(* Logix 5000 project; controller Pensador vendor 1 type 14 code 15 rev 20.11; software revision 20.04 *)

TASK MainTask (continuous, watchdog 500 ms) : MainProgram

MODULES
   Local : vendor 1 type 14 code 15 (SoftLogixController 2, rev 20.11)
      Ethernet : vendor 1 type 12 code 135 (SoftLogixVB 3, Ethernet 192.168.0.160, rev 20.1)
END_MODULES

VAR_GLOBAL   (* controller tags *)
   Acender_Led_Amarelo : BOOL := 1;
   Acender_Led_Azul : BOOL := 1;
   Acender_Led_Branco : BOOL := 1;
   Acender_Led_Transparente : BOOL;
   Acender_Led_Verde : BOOL := 1;
   Acender_Led_Vermelho : BOOL := 1;
   Acionamentos : DINT := 52;
   aguarde : BOOL;
   Alarme : DINT;
   Alinhador : STRING[20] := ([0] := 'Azul', [1] := 'Desliga_Azul', [2] := 'Vermelho', [3] := 'Desliga_Vermelho', [4] := 'Transparente', [5] := 'Desliga_Transparente', [6] := 'Amarelo', [7] := 'Desliga_Amarelo', [8] := 'Verde', [9] := 'Desliga_Verde');
   Botao_B01 : BOOL;
   Botao_B02 : BOOL := 1;
   Botao_B03 : BOOL;
   Botao_Pressionado : BOOL;
   Camera : STRING;
   CameraInt : DINT;
   Chamada_de_Voz : BOOL;
   Chave : SINT;
   Comparador : STRING := 'Ligar LED azul';
   Comparador2 : STRING := 'desligar led azul';
   Comparador3 : STRING := 'Ligar LED verde';
   Comparador4 : STRING := 'desligar led Verde';
   Comparador5 : STRING := 'Ligar LED branco';
   Comparador6 : STRING := 'desligar LED branco';
   Comparador7 : STRING := 'Ligar LED Amarelo';
   Comparador8 : STRING := 'desligar led Amarelo';
   Cont : DINT[10] := ([1] := 5);
   Conta_Acionamentos : COUNTER;
   ctus : COUNTER;
   D_0 : BOOL;
   D_2 : BOOL;
   D_3 : BOOL;
   D_5 : BOOL;
   D_6 : BOOL;
   Email_enviado : BOOL := 1;
   Entrada_D1 : BOOL;
   Entrada_D7 : BOOL;
   Entrada_D8 : BOOL;
   Enviar_Email : BOOL;
   Enviar_Mensagem : BOOL;
   Enviar_Mensagem_manualmente : BOOL;
   Enviar_SMS : BOOL;
   Enviar_SMS_Manualmente : BOOL := 1;
   Filtro : TIMER[10] := ([0].PRE := 500, [1].PRE := 500, [2].PRE := 500, [3].PRE := 500, [4].PRE := 500, [5].PRE := 500);
   FromEsp8266 : STRING;
   fromPLC : DINT := 2022;
   fromPython : DINT := 1984;
   Inicio : BOOL := 1;
   Input_0 : BOOL;
   Input_teste : DINT;
   Led_Amarelo : BOOL;   // This is for led Yelow Output D_5
   Led_Azul : BOOL;   // This is for led blue Output D_0
   Led_Transparente : BOOL;   // This is for led white Output D_3
   Led_Verde : BOOL;   // This is for led Green Output D_6
   Led_Vermelho : BOOL;   // This is for led red Output D_2
   Liga_Led_Amarelo : BOOL;
   Liga_Led_Azul : BOOL;
   Liga_Led_Green : BOOL;
   Liga_Led_Transparente : BOOL;
   Ligar : BOOL;
   Ligou : BOOL;
   Muthu : DINT := 88;
   Pisca_Lento : TIMER := (PRE := 1500);
   Pisca_Rapido : TIMER := (PRE := 1000);
   PLCout : STRING[10] := ([0] := 'Desliga_Vermelho', [1] := 'Input_010', [3] := '1985', [4] := '4', [5] := '4', [6] := '4');
   PlcToEsp8266 : DINT;
   PodeFalar : BOOL := 1;
   ProcessandoAudio : BOOL;
   Pulso : DINT := 31;
   Quant_Acionamentos : DINT := 158;
   Quantidade_Preditiva : DINT := 26;
   RecebeComando : STRING := 'maquiagem';
   receber : STRING;
   receive : DINT;
   ReceiveString : STRING := '568';
   Retem : TIMER;
   Retem_alarme : TIMER := (PRE := 10000, ACC := 10000);
   sendPLC : DINT;
   Shot : DINT := 1;
   Shot_Cont : BOOL := 1;
   SMS_enviado : BOOL := 1;
   Sorteio : DINT;
   Start : BOOL;
   Str : DINT[130] := ([1] := 1, [2] := 2, [3] := 3, [4] := 4, [5] := 5, [6] := 6, [7] := 7, [8] := 8, [9] := 9, [10] := 10, [11] := 11, [12] := 12, [13] := 13, [14] := 14, [15] := 15, [16] := 16, [17] := 17, [18] := 18, [19] := 19, [20] := 20, [21] := 21, [22] := 22, [23] := 23, [24] := 24, [25] := 25, [26] := 26, [27] := 27, [28] := 28, [29] := 29, [30] := 30, [31] := 31, [32] := 32);
   StringAvulsa : STRING[10] := ([0] := 'Input_000', [1] := 'Input_001', [2] := 'Input_010', [3] := 'Input_011', [4] := 'Input_100', [5] := 'Input_101', [6] := 'Input_110', [7] := 'Input_111');
   tagReceived : STRING;
   Tempo_devido : TIMER := (PRE := 15000, ACC := 15000);
   Temporizador : TIMER := (PRE := 10000);
   Testar_Alarme : BOOL;
   Teste_Alarme : DINT;
   Timer_1 : TIMER := (PRE := 1500);
   Timer_2 : TIMER := (PRE := 1500);
   Whatsapp_MSG : DINT := 52;
   Zerar_Contadores : BOOL;
END_VAR

PROGRAM MainProgram   (* main routine MainRoutine *)

ROUTINE _alarmes   (* ladder *)
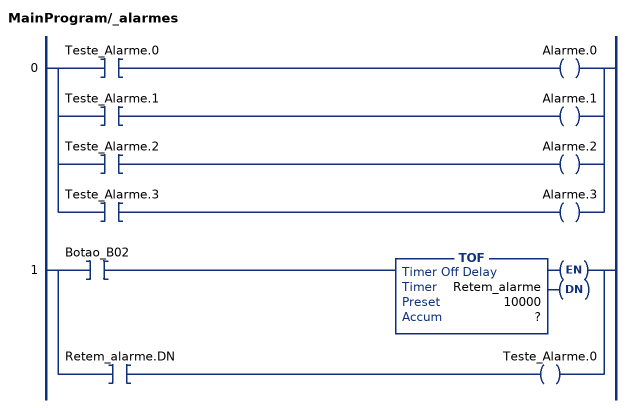
   0: [XIC(Teste_Alarme.0) OTE(Alarme.0) ,XIC(Teste_Alarme.1) OTE(Alarme.1) ,XIC(Teste_Alarme.2) OTE(Alarme.2) ,XIC(Teste_Alarme.3) OTE(Alarme.3) ];
   1: [XIC(Botao_B02) TOF(Retem_alarme,?,?) ,XIC(Retem_alarme.DN) OTE(Teste_Alarme.0) ];
END_ROUTINE

ROUTINE _Dois_Modulos   (* ladder *)
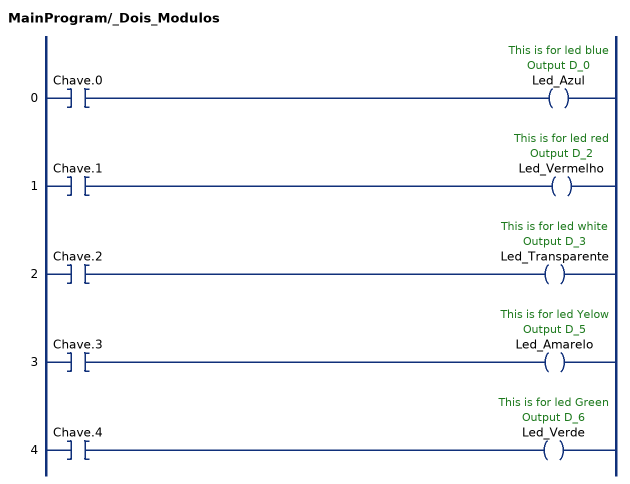
   0: XIC(Chave.0)OTE(Led_Azul);
   1: XIC(Chave.1)OTE(Led_Vermelho);
   2: XIC(Chave.2)OTE(Led_Transparente);
   3: XIC(Chave.3)OTE(Led_Amarelo);
   4: XIC(Chave.4)OTE(Led_Verde);
END_ROUTINE

ROUTINE Acionamento_INPUTS   (* ladder *)
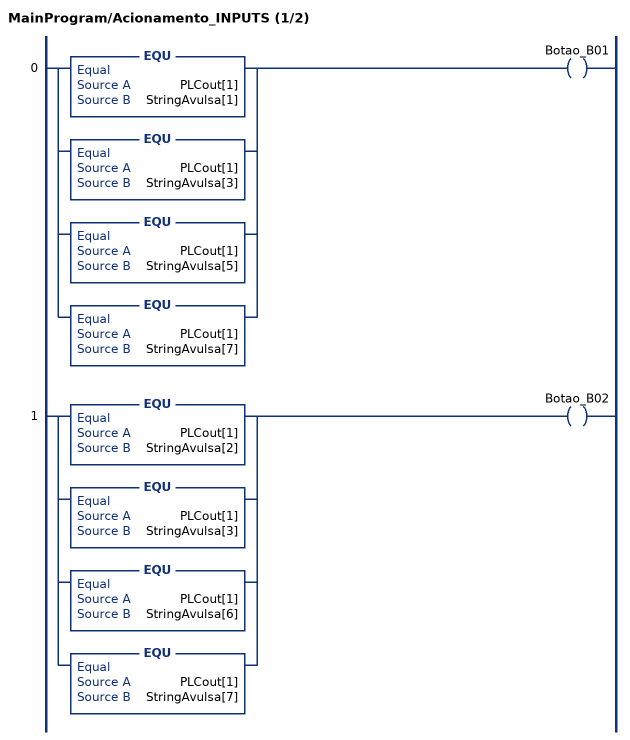
   0: [EQU(PLCout[1],StringAvulsa[1]) ,EQU(PLCout[1],StringAvulsa[3]) ,EQU(PLCout[1],StringAvulsa[5]) ,EQU(PLCout[1],StringAvulsa[7]) ]OTE(Botao_B01);
   1: [EQU(PLCout[1],StringAvulsa[2]) ,EQU(PLCout[1],StringAvulsa[3]) ,EQU(PLCout[1],StringAvulsa[6]) ,EQU(PLCout[1],StringAvulsa[7]) ]OTE(Botao_B02);
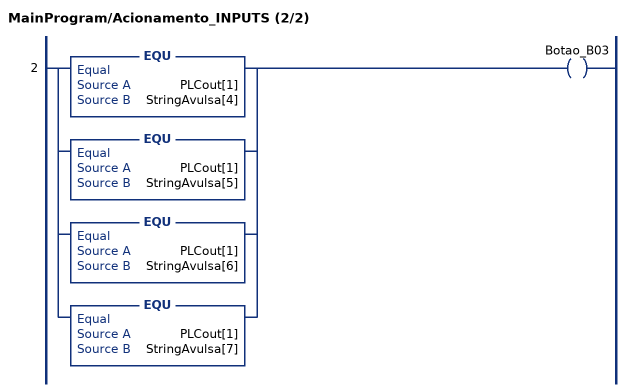
   2: [EQU(PLCout[1],StringAvulsa[4]) ,EQU(PLCout[1],StringAvulsa[5]) ,EQU(PLCout[1],StringAvulsa[6]) ,EQU(PLCout[1],StringAvulsa[7]) ]OTE(Botao_B03);
END_ROUTINE

ROUTINE Acionamento_OUTPUTS   (* ladder *)
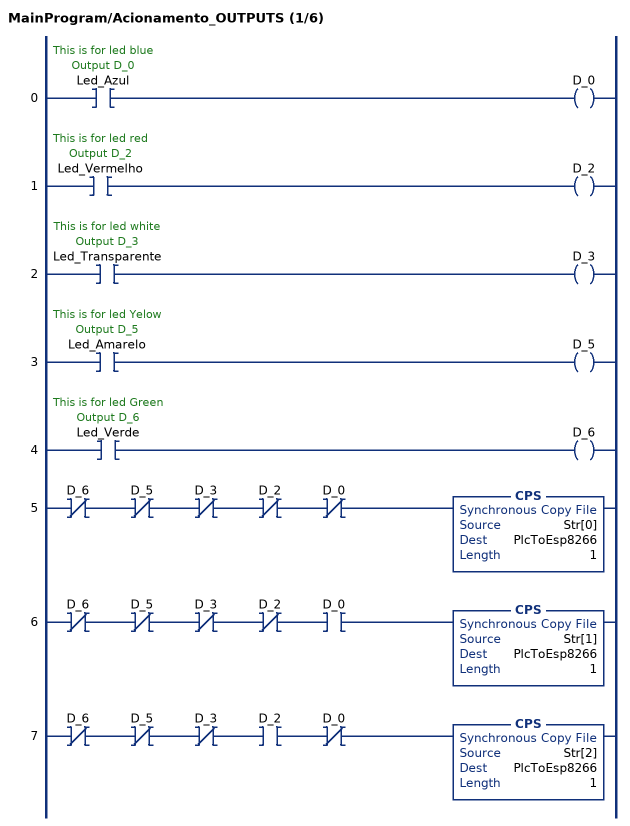
   0: XIC(Led_Azul)OTE(D_0);
   1: XIC(Led_Vermelho)OTE(D_2);
   2: XIC(Led_Transparente)OTE(D_3);
   3: XIC(Led_Amarelo)OTE(D_5);
   4: XIC(Led_Verde)OTE(D_6);
   5: XIO(D_6)XIO(D_5)XIO(D_3)XIO(D_2)XIO(D_0)CPS(Str[0],PlcToEsp8266,1);
   6: XIO(D_6)XIO(D_5)XIO(D_3)XIO(D_2)XIC(D_0)CPS(Str[1],PlcToEsp8266,1);
   7: XIO(D_6)XIO(D_5)XIO(D_3)XIC(D_2)XIO(D_0)CPS(Str[2],PlcToEsp8266,1);
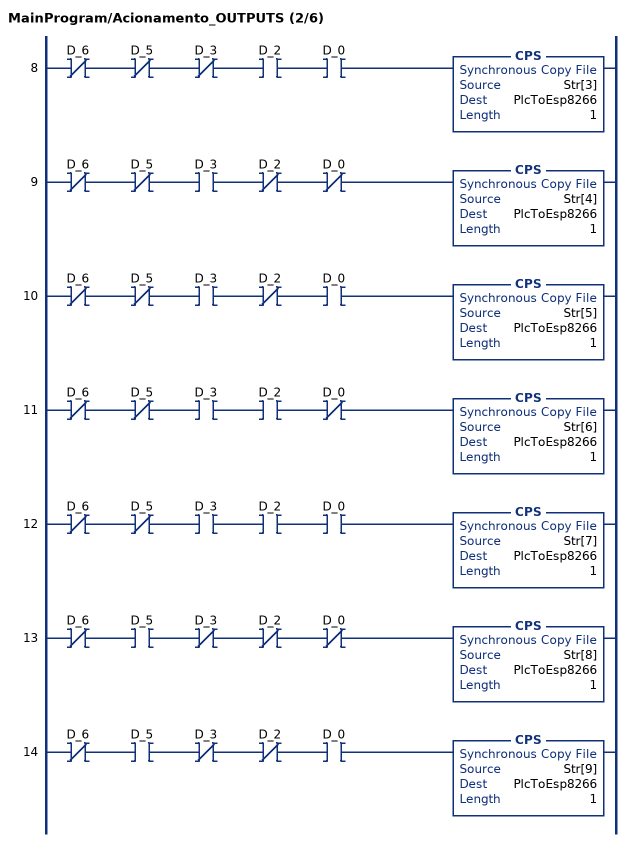
   8: XIO(D_6)XIO(D_5)XIO(D_3)XIC(D_2)XIC(D_0)CPS(Str[3],PlcToEsp8266,1);
   9: XIO(D_6)XIO(D_5)XIC(D_3)XIO(D_2)XIO(D_0)CPS(Str[4],PlcToEsp8266,1);
   10: XIO(D_6)XIO(D_5)XIC(D_3)XIO(D_2)XIC(D_0)CPS(Str[5],PlcToEsp8266,1);
   11: XIO(D_6)XIO(D_5)XIC(D_3)XIC(D_2)XIO(D_0)CPS(Str[6],PlcToEsp8266,1);
   12: XIO(D_6)XIO(D_5)XIC(D_3)XIC(D_2)XIC(D_0)CPS(Str[7],PlcToEsp8266,1);
   13: XIO(D_6)XIC(D_5)XIO(D_3)XIO(D_2)XIO(D_0)CPS(Str[8],PlcToEsp8266,1);
   14: XIO(D_6)XIC(D_5)XIO(D_3)XIO(D_2)XIC(D_0)CPS(Str[9],PlcToEsp8266,1);
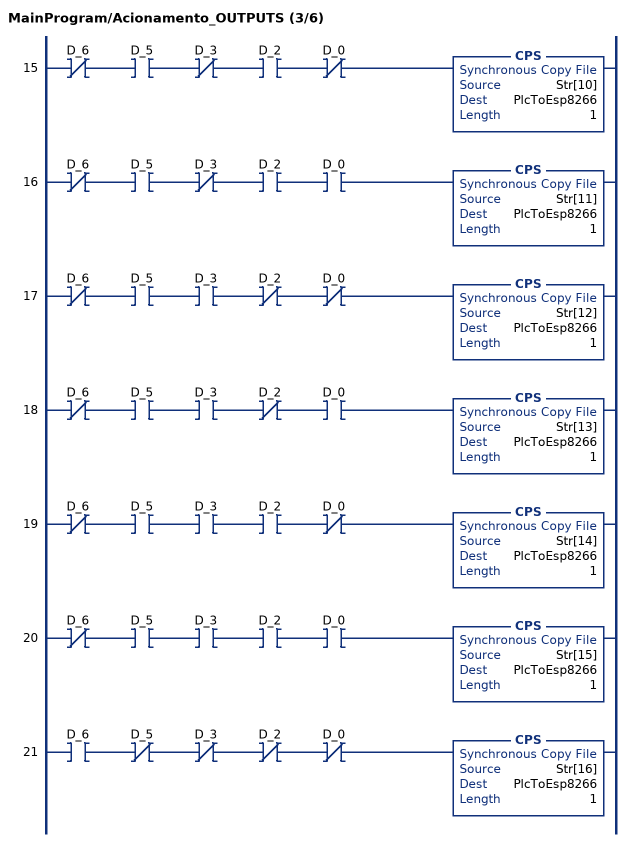
   15: XIO(D_6)XIC(D_5)XIO(D_3)XIC(D_2)XIO(D_0)CPS(Str[10],PlcToEsp8266,1);
   16: XIO(D_6)XIC(D_5)XIO(D_3)XIC(D_2)XIC(D_0)CPS(Str[11],PlcToEsp8266,1);
   17: XIO(D_6)XIC(D_5)XIC(D_3)XIO(D_2)XIO(D_0)CPS(Str[12],PlcToEsp8266,1);
   18: XIO(D_6)XIC(D_5)XIC(D_3)XIO(D_2)XIC(D_0)CPS(Str[13],PlcToEsp8266,1);
   19: XIO(D_6)XIC(D_5)XIC(D_3)XIC(D_2)XIO(D_0)CPS(Str[14],PlcToEsp8266,1);
   20: XIO(D_6)XIC(D_5)XIC(D_3)XIC(D_2)XIC(D_0)CPS(Str[15],PlcToEsp8266,1);
   21: XIC(D_6)XIO(D_5)XIO(D_3)XIO(D_2)XIO(D_0)CPS(Str[16],PlcToEsp8266,1);
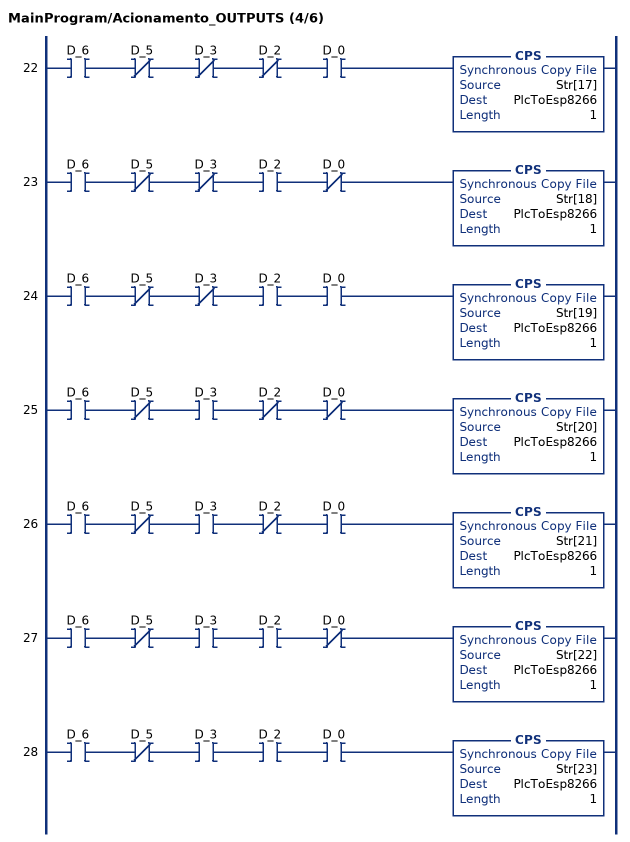
   22: XIC(D_6)XIO(D_5)XIO(D_3)XIO(D_2)XIC(D_0)CPS(Str[17],PlcToEsp8266,1);
   23: XIC(D_6)XIO(D_5)XIO(D_3)XIC(D_2)XIO(D_0)CPS(Str[18],PlcToEsp8266,1);
   24: XIC(D_6)XIO(D_5)XIO(D_3)XIC(D_2)XIC(D_0)CPS(Str[19],PlcToEsp8266,1);
   25: XIC(D_6)XIO(D_5)XIC(D_3)XIO(D_2)XIO(D_0)CPS(Str[20],PlcToEsp8266,1);
   26: XIC(D_6)XIO(D_5)XIC(D_3)XIO(D_2)XIC(D_0)CPS(Str[21],PlcToEsp8266,1);
   27: XIC(D_6)XIO(D_5)XIC(D_3)XIC(D_2)XIO(D_0)CPS(Str[22],PlcToEsp8266,1);
   28: XIC(D_6)XIO(D_5)XIC(D_3)XIC(D_2)XIC(D_0)CPS(Str[23],PlcToEsp8266,1);
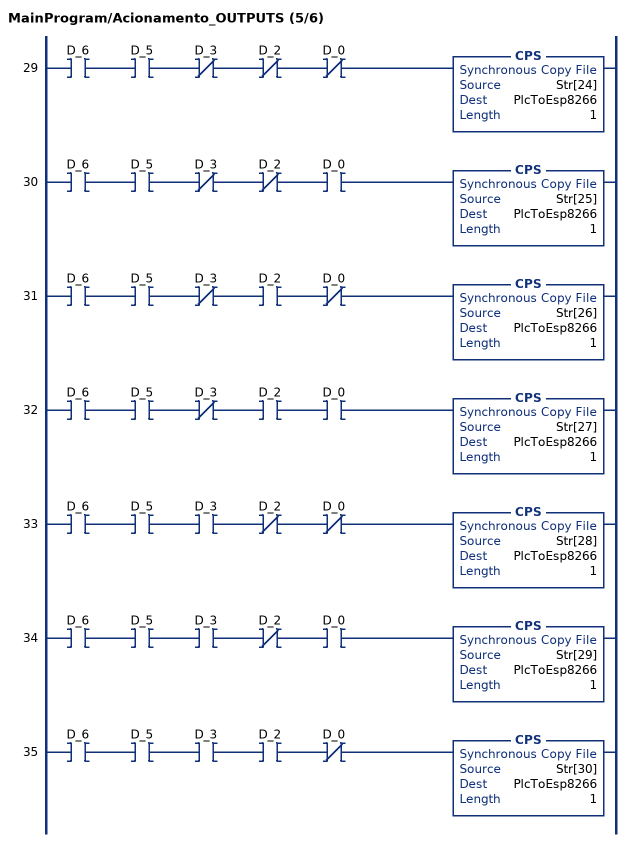
   29: XIC(D_6)XIC(D_5)XIO(D_3)XIO(D_2)XIO(D_0)CPS(Str[24],PlcToEsp8266,1);
   30: XIC(D_6)XIC(D_5)XIO(D_3)XIO(D_2)XIC(D_0)CPS(Str[25],PlcToEsp8266,1);
   31: XIC(D_6)XIC(D_5)XIO(D_3)XIC(D_2)XIO(D_0)CPS(Str[26],PlcToEsp8266,1);
   32: XIC(D_6)XIC(D_5)XIO(D_3)XIC(D_2)XIC(D_0)CPS(Str[27],PlcToEsp8266,1);
   33: XIC(D_6)XIC(D_5)XIC(D_3)XIO(D_2)XIO(D_0)CPS(Str[28],PlcToEsp8266,1);
   34: XIC(D_6)XIC(D_5)XIC(D_3)XIO(D_2)XIC(D_0)CPS(Str[29],PlcToEsp8266,1);
   35: XIC(D_6)XIC(D_5)XIC(D_3)XIC(D_2)XIO(D_0)CPS(Str[30],PlcToEsp8266,1);
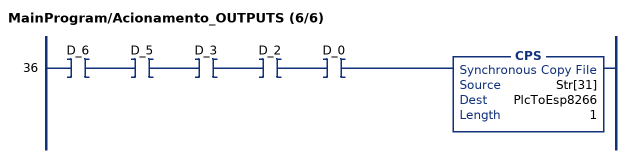
   36: XIC(D_6)XIC(D_5)XIC(D_3)XIC(D_2)XIC(D_0)CPS(Str[31],PlcToEsp8266,1);
END_ROUTINE

ROUTINE Bot_Whatsapp   (* ladder *)
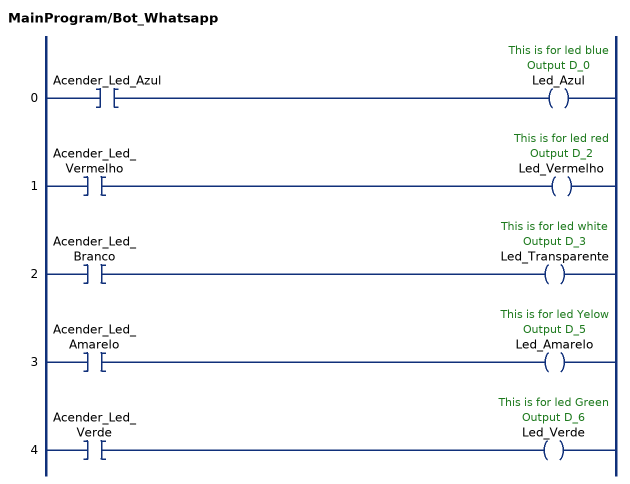
   0: XIC(Acender_Led_Azul)OTE(Led_Azul);
   1: XIC(Acender_Led_Vermelho)OTE(Led_Vermelho);
   2: XIC(Acender_Led_Branco)OTE(Led_Transparente);
   3: XIC(Acender_Led_Amarelo)OTE(Led_Amarelo);
   4: XIC(Acender_Led_Verde)OTE(Led_Verde);
END_ROUTINE

ROUTINE Camera   (* ladder *)
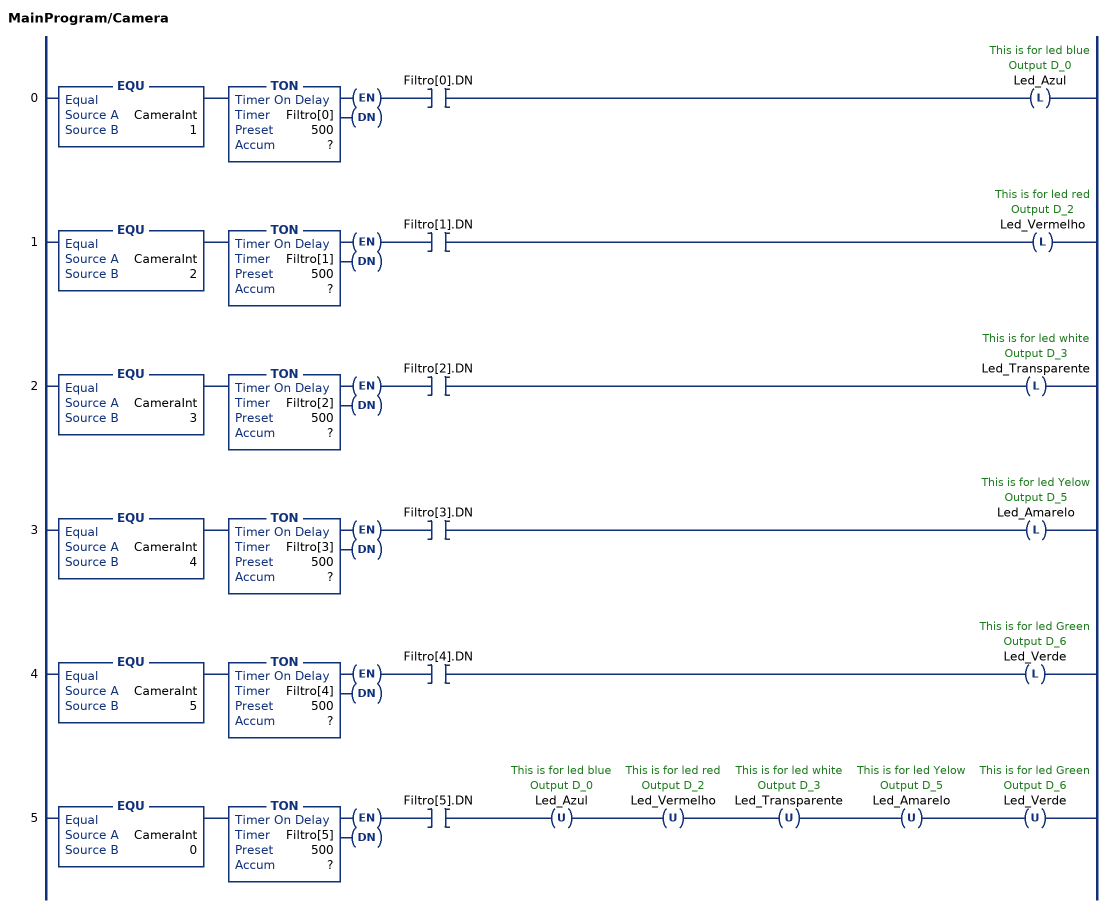
   0: EQU(CameraInt,1)TON(Filtro[0],?,?)XIC(Filtro[0].DN)OTL(Led_Azul);
   1: EQU(CameraInt,2)TON(Filtro[1],?,?)XIC(Filtro[1].DN)OTL(Led_Vermelho);
   2: EQU(CameraInt,3)TON(Filtro[2],?,?)XIC(Filtro[2].DN)OTL(Led_Transparente);
   3: EQU(CameraInt,4)TON(Filtro[3],?,?)XIC(Filtro[3].DN)OTL(Led_Amarelo);
   4: EQU(CameraInt,5)TON(Filtro[4],?,?)XIC(Filtro[4].DN)OTL(Led_Verde);
   5: EQU(CameraInt,0)TON(Filtro[5],?,?)XIC(Filtro[5].DN)OTU(Led_Azul)OTU(Led_Vermelho)OTU(Led_Transparente)OTU(Led_Amarelo)OTU(Led_Verde);
END_ROUTINE

ROUTINE Comando_De_Voz   (* ladder *)
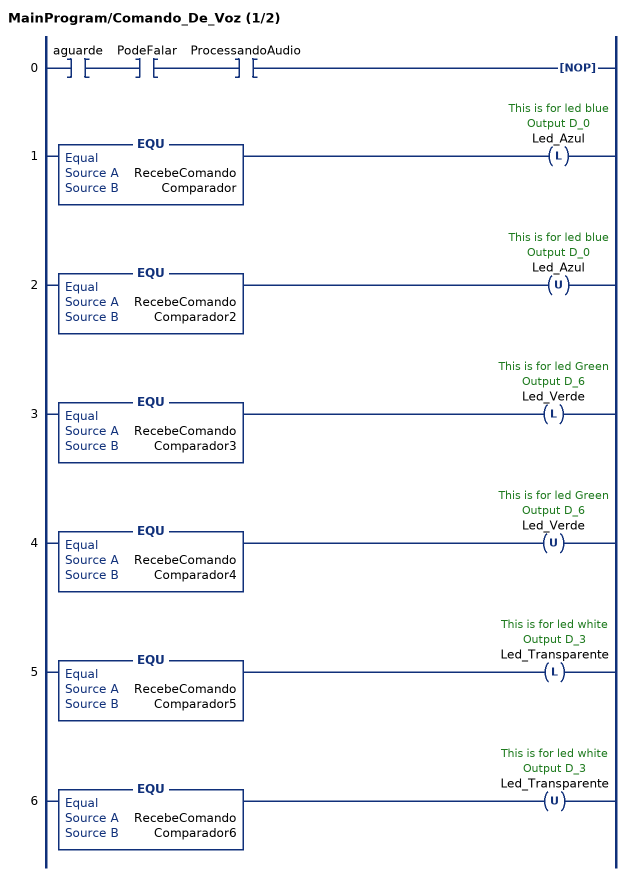
   0: XIC(aguarde)XIC(PodeFalar)XIC(ProcessandoAudio)NOP();
   1: EQU(RecebeComando,Comparador)OTL(Led_Azul);
   2: EQU(RecebeComando,Comparador2)OTU(Led_Azul);
   3: EQU(RecebeComando,Comparador3)OTL(Led_Verde);
   4: EQU(RecebeComando,Comparador4)OTU(Led_Verde);
   5: EQU(RecebeComando,Comparador5)OTL(Led_Transparente);
   6: EQU(RecebeComando,Comparador6)OTU(Led_Transparente);
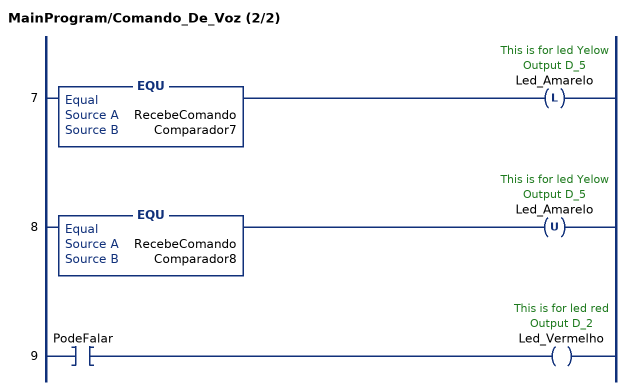
   7: EQU(RecebeComando,Comparador7)OTL(Led_Amarelo);
   8: EQU(RecebeComando,Comparador8)OTU(Led_Amarelo);
   9: XIC(PodeFalar)OTE(Led_Vermelho);
END_ROUTINE

ROUTINE Comandos   (* ladder *)
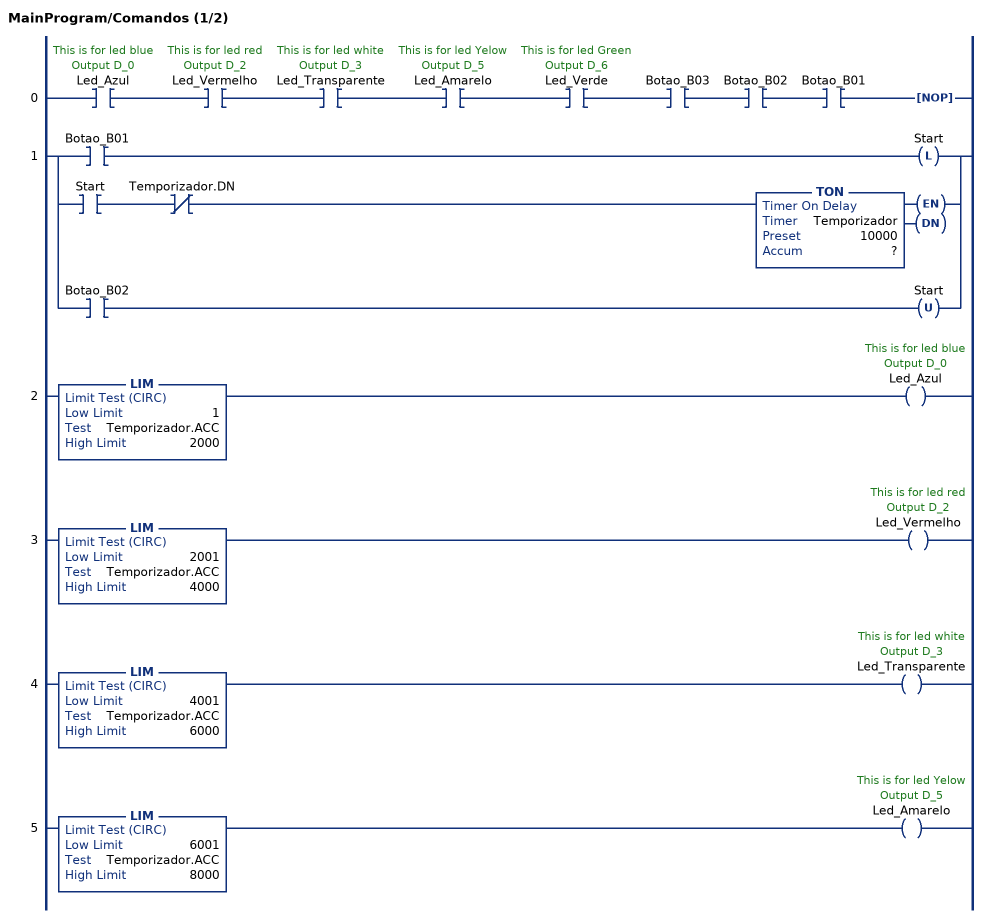
   0: XIC(Led_Azul)XIC(Led_Vermelho)XIC(Led_Transparente)XIC(Led_Amarelo)XIC(Led_Verde)XIC(Botao_B03)XIC(Botao_B02)XIC(Botao_B01)NOP();
   1: [XIC(Botao_B01) OTL(Start) ,XIC(Start) XIO(Temporizador.DN) TON(Temporizador,?,?) ,XIC(Botao_B02) OTU(Start) ];
   2: LIM(1,Temporizador.ACC,2000)OTE(Led_Azul);
   3: LIM(2001,Temporizador.ACC,4000)OTE(Led_Vermelho);
   4: LIM(4001,Temporizador.ACC,6000)OTE(Led_Transparente);
   5: LIM(6001,Temporizador.ACC,8000)OTE(Led_Amarelo);
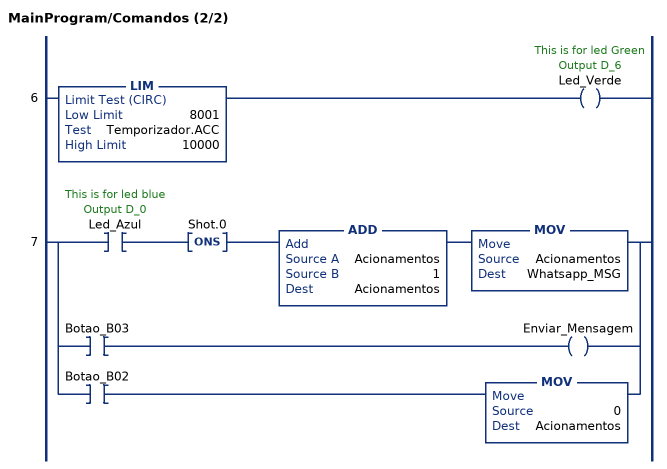
   6: LIM(8001,Temporizador.ACC,10000)OTE(Led_Verde);
   7: [XIC(Led_Azul) ONS(Shot.0) ADD(Acionamentos,1,Acionamentos) MOV(Acionamentos,Whatsapp_MSG) ,XIC(Botao_B03) OTE(Enviar_Mensagem) ,XIC(Botao_B02) MOV(0,Acionamentos) ];
END_ROUTINE

ROUTINE Email   (* ladder *)
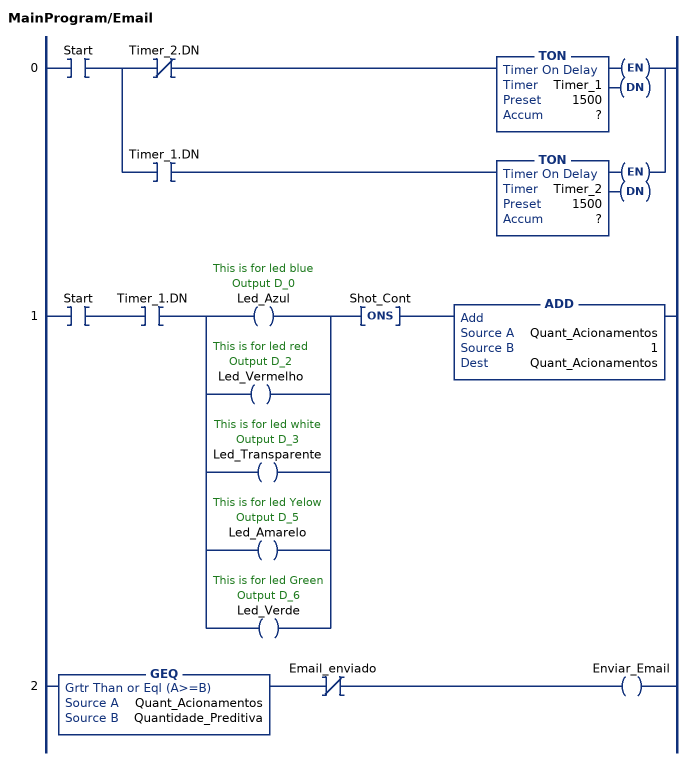
   0: XIC(Start)[XIO(Timer_2.DN) TON(Timer_1,?,?) ,XIC(Timer_1.DN) TON(Timer_2,?,?) ];
   1: XIC(Start)XIC(Timer_1.DN)[OTE(Led_Azul) ,OTE(Led_Vermelho) ,OTE(Led_Transparente) ,OTE(Led_Amarelo) ,OTE(Led_Verde) ]ONS(Shot_Cont)ADD(Quant_Acionamentos,1,Quant_Acionamentos);
   2: GEQ(Quant_Acionamentos,Quantidade_Preditiva)XIO(Email_enviado)OTE(Enviar_Email);
END_ROUTINE

ROUTINE india   (* ladder *)
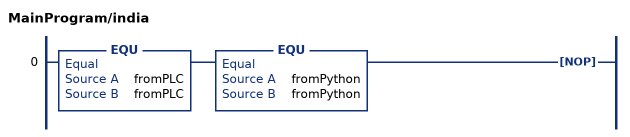
   0: EQU(fromPLC,fromPLC)EQU(fromPython,fromPython)NOP();
END_ROUTINE

ROUTINE Ligacao   (* ladder *)
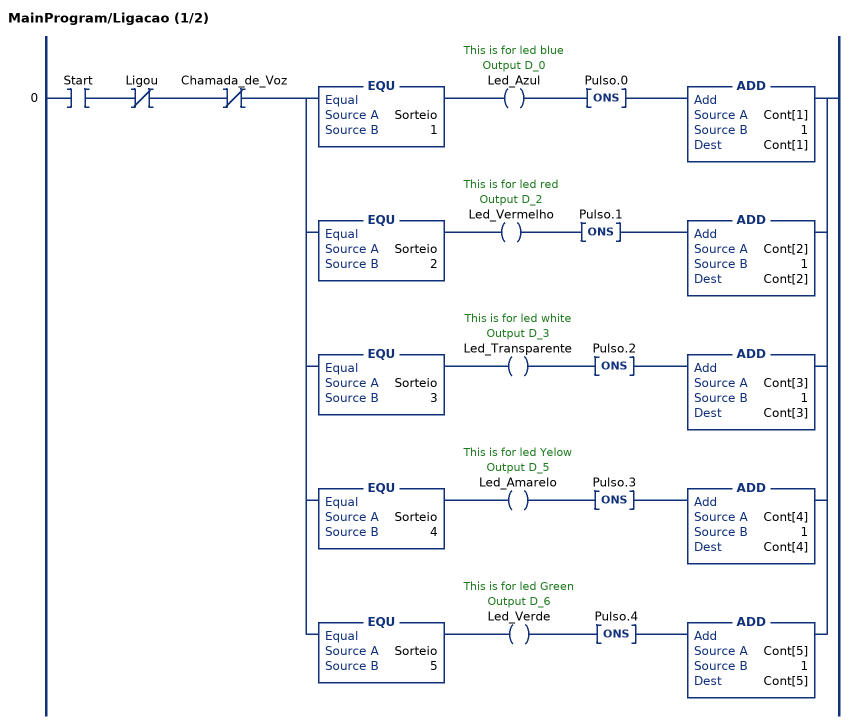
   0: XIC(Start)XIO(Ligou)XIO(Chamada_de_Voz)[EQU(Sorteio,1) OTE(Led_Azul) ONS(Pulso.0) ADD(Cont[1],1,Cont[1]) ,EQU(Sorteio,2) OTE(Led_Vermelho) ONS(Pulso.1) ADD(Cont[2],1,Cont[2]) ,EQU(Sorteio,3) OTE(Led_Transparente) ONS(Pulso.2) ADD(Cont[3],1,Cont[3]) ,EQU(Sorteio,4) OTE(Led_Amarelo) ONS(Pulso.3) ADD(Cont[4],1,Cont[4]) ,EQU(Sorteio,5) OTE(Led_Verde) ONS(Pulso.4) ADD(Cont[5],1,Cont[5]) ];
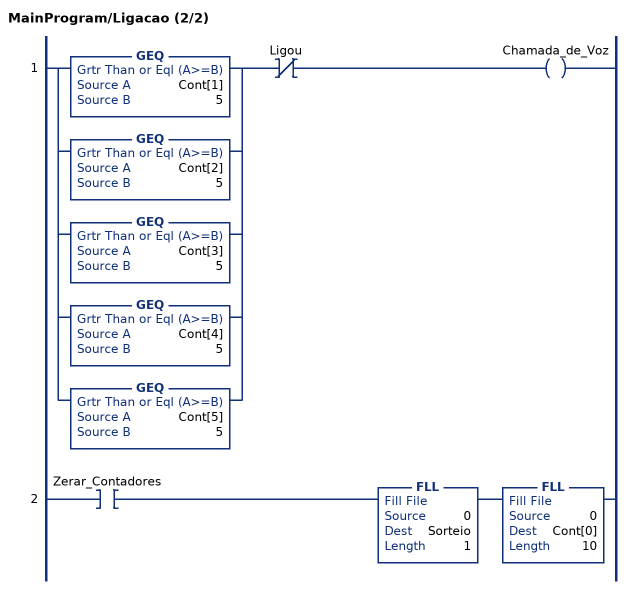
   1: [GEQ(Cont[1],5) ,GEQ(Cont[2],5) ,GEQ(Cont[3],5) ,GEQ(Cont[4],5) ,GEQ(Cont[5],5) ]XIO(Ligou)OTE(Chamada_de_Voz);
   2: XIC(Zerar_Contadores)FLL(0,Sorteio,1)FLL(0,Cont[0],10);
END_ROUTINE

ROUTINE MainRoutine   (* ladder *)
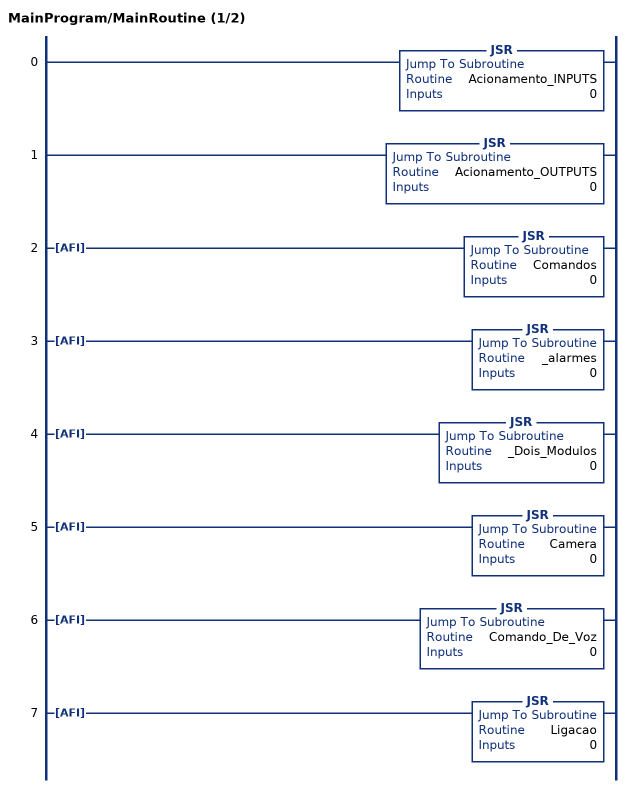
   0: JSR(Acionamento_INPUTS,0);
   1: JSR(Acionamento_OUTPUTS,0);
   2: AFI()JSR(Comandos,0);
   3: AFI()JSR(_alarmes,0);
   4: AFI()JSR(_Dois_Modulos,0);
   5: AFI()JSR(Camera,0);
   6: AFI()JSR(Comando_De_Voz,0);
   7: AFI()JSR(Ligacao,0);
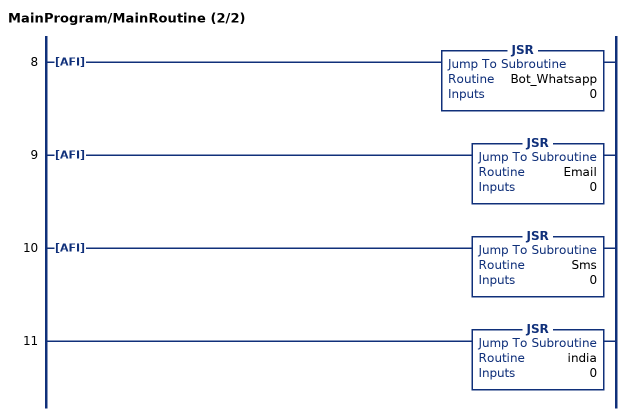
   8: AFI()JSR(Bot_Whatsapp,0);
   9: AFI()JSR(Email,0);
   10: AFI()JSR(Sms,0);
   11: JSR(india,0);
END_ROUTINE

ROUTINE Sms   (* ladder *)
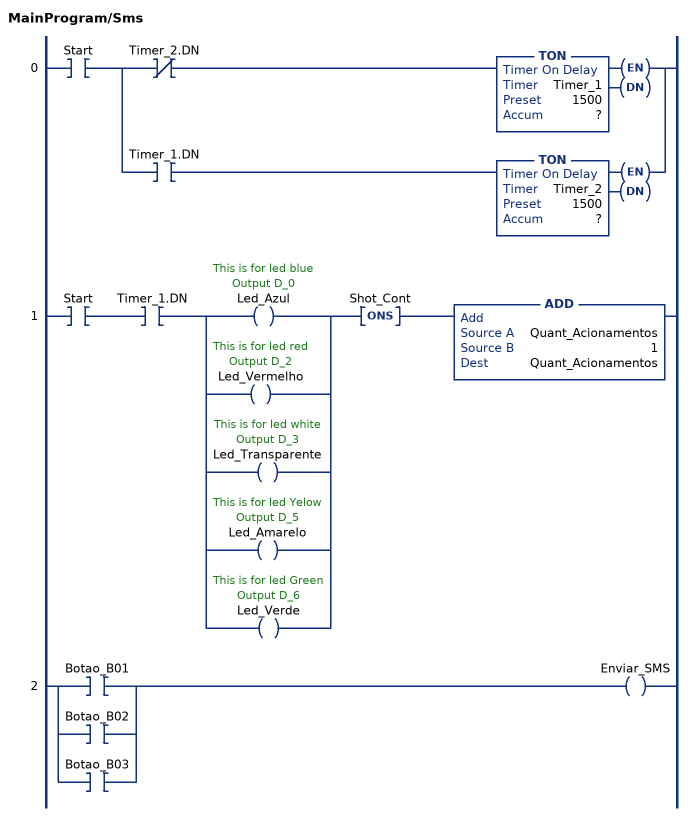
   0: XIC(Start)[XIO(Timer_2.DN) TON(Timer_1,?,?) ,XIC(Timer_1.DN) TON(Timer_2,?,?) ];
   1: XIC(Start)XIC(Timer_1.DN)[OTE(Led_Azul) ,OTE(Led_Vermelho) ,OTE(Led_Transparente) ,OTE(Led_Amarelo) ,OTE(Led_Verde) ]ONS(Shot_Cont)ADD(Quant_Acionamentos,1,Quant_Acionamentos);
   2: [XIC(Botao_B01) ,XIC(Botao_B02) ,XIC(Botao_B03) ]OTE(Enviar_SMS);
END_ROUTINE
END_PROGRAM
